// TIA Portal V17 export
// export: Created 2024-09-15T12:29:52.0715194Z, ExportSetting WithDefaults, DisplayName Totally Integrated Automation Portal, DisplayVersion V17, DisplayName TIA Portal Openness, DisplayVersion V17, DisplayName TIA Portal Version Control Interface, DisplayVersion V17, DisplayName STEP 7 Professional, DisplayVersion V17, DisplayName STEP 7 Safety, DisplayVersion V17, DisplayName WinCC Professional, DisplayVersion V17
DATA_BLOCK "gtyp_HBW"   // DB17
TITLE = Global DB HBW
{ S7_Optimized_Access := 'TRUE' }
AUTHOR : A.Schaefer
VERSION : 0.0
// stored: AutoNumber true, DBAccessibleFromOPCUA true, DBAccessibleFromWebserver true, InstanceOfName typ_HBW, InstanceOfType UDT, IsOnlyStoredInLoadMemory false, IsWriteProtectedInAS false
"typ_HBW"
   // VAR RETAIN
   //    x_Start_Park_Position : Bool;
   //    x_Park_Position_Reached : Bool;
   //    x_HBW_PickedUp_Accepted : Bool;
   //    x_HBW_Discards_Accepted : Bool;
   //    x_HBW_PickUp_Ready : Bool;
   //    x_HBW_Container_Available : Bool;
   //    x_Error : Bool;
   //    s_ErrorMessage : String;
   //    di_PosBelt_Horizontal : DInt := 18;
   //    di_PosBelt_Vertical : DInt := 2800;
   //    di_Offset_Pos_Belt_Vertical : DInt := 370;
   //    di_PosRack_A1_Horizontal : DInt := 2870;
   //    di_PosRack_A1_Vertical : DInt := 400;
   //    di_PosRack_B2_Horizontal : DInt := 5215;
   //    di_PosRack_B2_Vertical : DInt := 1750;
   //    di_PosRack_C3_Horizontal : DInt := 7560;
   //    di_PosRack_C3_Vertical : DInt := 3300;
   //    di_Offset_Pos_Rack_Vertical : DInt := 370;
   //    di_Pos_Park_Horizontal : DInt := 600;
   //    di_Pos_Park_Vertical : DInt := 3200;
   //    i_PWM_ConveyorBelt : Int;
   //    i_PWM_Cantilever : Int := 1000;
   //    Workpiece : "typ_Workpiece";
   //    History : Array[1..20] of "typ_History";
   //    Rack_Pos : Array[1..3, 1..3] of "typ_Rack_Pos";
   //    Rack_Workpiece : Array[1..3, 1..3] of "typ_Workpiece";
   //    Rack_History : Array[1..3, 1..3] of "typ_Rack_History";
   //    Horizontal_Axis : "typ_Axis";
   //    Vertical_Axis : "typ_Axis";
   //    i_Red_Available { S7_SetPoint := 'True'} : Int;
   //    i_Blue_Available : Int;
   //    i_White_Available : Int;
   //    di_Offset_Actual_Pickup : DInt := 150;
   // END_VAR
BEGIN
   Rack_Pos[1,1].di_PosRack_Horizontal := 2870;
   Rack_Pos[1,2].di_PosRack_Horizontal := 5200;
   Rack_Pos[1,3].di_PosRack_Horizontal := 7550;
   Rack_Pos[2,1].di_PosRack_Horizontal := 2870;
   Rack_Pos[2,2].di_PosRack_Horizontal := 5200;
   Rack_Pos[2,3].di_PosRack_Horizontal := 7550;
   Rack_Pos[3,1].di_PosRack_Horizontal := 2870;
   Rack_Pos[3,2].di_PosRack_Horizontal := 5200;
   Rack_Pos[3,3].di_PosRack_Horizontal := 7550;
   Rack_Pos[1,1..3].di_PosRack_Vertical := 400;
   Rack_Pos[2,1..3].di_PosRack_Vertical := 1750;
   Rack_Pos[3,1..3].di_PosRack_Vertical := 3150;
   Rack_Workpiece[1,1..3].s_id := '0';
   Rack_Workpiece[2,1..3].s_id := '0';
   Rack_Workpiece[3,1..3].s_id := '0';
   Horizontal_Axis.i_PWM := -1;
   Horizontal_Axis.Config.di_Pos_Soft_Switch := 7900;
   Horizontal_Axis.Config.di_Pos_Window := 15;
   Vertical_Axis.i_PWM := -1;
   Vertical_Axis.Config.di_Pos_Soft_Switch := 3350;
   Vertical_Axis.Config.di_Pos_Window := 15;
END_DATA_BLOCK
